FUNCTION_BLOCK EL3064
VAR
	_io : EL3xx4_Data;
	{attribute addProperty Name "WcState"}
	_wcState : WcStateInputToggle;
	{attribute addProperty Name "Info data"}
	_infoData : InfoDataAds;
END_VAR

PROPERTY IO : REFERENCE TO EL3xx4_Data
GET
IO REF= _io;
END_GET
END_PROPERTY

PROPERTY WcState : REFERENCE TO WcStateInputToggle
GET
WcState REF= _wcState;
END_GET
END_PROPERTY

END_FUNCTION_BLOCK

(* stored: Version 1.1.0.1, ProductVersion 3.1.4024.9
   POU EL3064: Id {6441c201-0b06-0673-1d03-85b68e4af030}, SpecialFunc None
   Property IO: Id {ce279c4b-0f34-0d28-31a7-d16e38a595e2}
   Get Get: Id {5761d3d6-634e-08f0-1fb8-b3981376e718}
   Property WcState: Id {39c0d7b2-9284-0338-0ac1-b2ac5139424f}
   Get Get: Id {caaa6102-de72-08dd-375f-211fc322b0c9} *)
